SUBAPPLICATION Heckschieber (* Subapplication Type *)
  (* Standard: 61499-2 *)
  (* Version 1.0, 2023-01-29, Franz *)
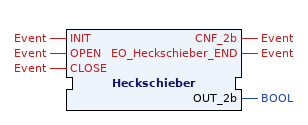
  EVENT_INPUT
    INIT;
    OPEN;
    CLOSE;
  END_EVENT
  EVENT_OUTPUT
    CNF_2b;
    EO_Heckschieber_END;
  END_EVENT
  VAR_OUTPUT
    OUT_2b : BOOL;
  END_VAR
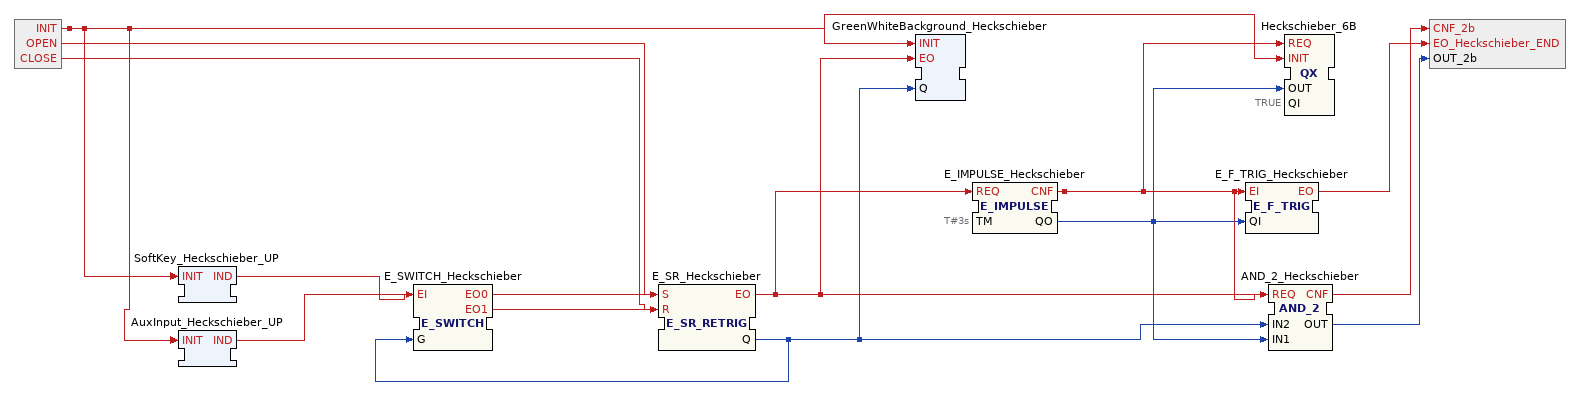
  FBS
    E_F_TRIG_Heckschieber : E_F_TRIG;
    Heckschieber_6B : QX(QI := TRUE);
    E_SR_Heckschieber : E_SR_RETRIG;
    E_SWITCH_Heckschieber : E_SWITCH;
    AND_2_Heckschieber : AND_2;
    E_IMPULSE_Heckschieber : E_IMPULSE(TM := T#3s);
  END_FBS
  SUBAPPLICATION AuxInput_Heckschieber_UP
    EVENT_INPUT
      INIT;
    END_EVENT
    EVENT_OUTPUT
      IND;
    END_EVENT
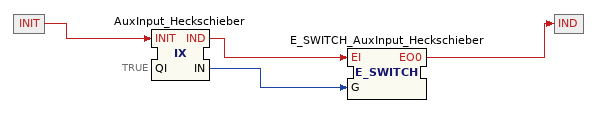
    FBS
      E_SWITCH_AuxInput_Heckschieber : E_SWITCH;
      AuxInput_Heckschieber : IX(QI := TRUE);
    END_FBS
    EVENT_CONNECTIONS
      AuxInput_Heckschieber.IND TO E_SWITCH_AuxInput_Heckschieber.EI;
      INIT TO AuxInput_Heckschieber.INIT;
      E_SWITCH_AuxInput_Heckschieber.EO0 TO IND;
    END_CONNECTIONS
    DATA_CONNECTIONS
      AuxInput_Heckschieber.IN TO E_SWITCH_AuxInput_Heckschieber.G;
    END_CONNECTIONS
  END_SUBAPPLICATION
  SUBAPPLICATION GreenWhiteBackground_Heckschieber
    EVENT_INPUT
      INIT;
      EO;
    END_EVENT
    VAR_INPUT
      Q : BOOL;
    END_VAR
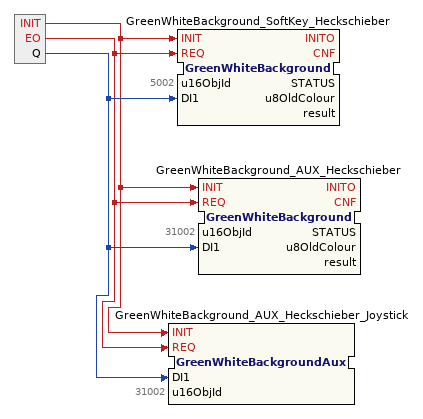
    FBS
      GreenWhiteBackground_SoftKey_Heckschieber : GreenWhiteBackground(u16ObjId := 5002);
      GreenWhiteBackground_AUX_Heckschieber : GreenWhiteBackground(u16ObjId := 31002);
      GreenWhiteBackground_AUX_Heckschieber_Joystick : GreenWhiteBackgroundAux(u16ObjId := 31002);
    END_FBS
    EVENT_CONNECTIONS
      INIT TO GreenWhiteBackground_SoftKey_Heckschieber.INIT;
      EO TO GreenWhiteBackground_SoftKey_Heckschieber.REQ;
      INIT TO GreenWhiteBackground_AUX_Heckschieber.INIT;
      EO TO GreenWhiteBackground_AUX_Heckschieber.REQ;
      INIT TO GreenWhiteBackground_AUX_Heckschieber_Joystick.INIT;
      EO TO GreenWhiteBackground_AUX_Heckschieber_Joystick.REQ;
    END_CONNECTIONS
    DATA_CONNECTIONS
      Q TO GreenWhiteBackground_SoftKey_Heckschieber.DI1;
      Q TO GreenWhiteBackground_AUX_Heckschieber.DI1;
      Q TO GreenWhiteBackground_AUX_Heckschieber_Joystick.DI1;
    END_CONNECTIONS
  END_SUBAPPLICATION
  SUBAPPLICATION SoftKey_Heckschieber_UP
    EVENT_INPUT
      INIT;
    END_EVENT
    EVENT_OUTPUT
      IND;
    END_EVENT
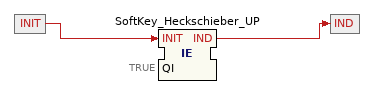
    FBS
      SoftKey_Heckschieber_UP : IE(QI := TRUE);
    END_FBS
    EVENT_CONNECTIONS
      INIT TO SoftKey_Heckschieber_UP.INIT;
      SoftKey_Heckschieber_UP.IND TO IND;
    END_CONNECTIONS
  END_SUBAPPLICATION
  EVENT_CONNECTIONS
    E_IMPULSE_Heckschieber.CNF TO E_F_TRIG_Heckschieber.EI;
    E_IMPULSE_Heckschieber.CNF TO Heckschieber_6B.REQ;
    E_SWITCH_Heckschieber.EO0 TO E_SR_Heckschieber.S;
    E_SWITCH_Heckschieber.EO1 TO E_SR_Heckschieber.R;
    E_SR_Heckschieber.EO TO AND_2_Heckschieber.REQ;
    E_SR_Heckschieber.EO TO E_IMPULSE_Heckschieber.REQ;
    E_IMPULSE_Heckschieber.CNF TO AND_2_Heckschieber.REQ;
    OPEN TO E_SR_Heckschieber.S;
    CLOSE TO E_SR_Heckschieber.R;
    AND_2_Heckschieber.CNF TO CNF_2b;
    E_F_TRIG_Heckschieber.EO TO EO_Heckschieber_END;
    AuxInput_Heckschieber_UP.IND TO E_SWITCH_Heckschieber.EI;
    INIT TO AuxInput_Heckschieber_UP.INIT;
    INIT TO GreenWhiteBackground_Heckschieber.INIT;
    E_SR_Heckschieber.EO TO GreenWhiteBackground_Heckschieber.EO;
    INIT TO SoftKey_Heckschieber_UP.INIT;
    SoftKey_Heckschieber_UP.IND TO E_SWITCH_Heckschieber.EI;
    INIT TO Heckschieber_6B.INIT;
  END_CONNECTIONS
  DATA_CONNECTIONS
    E_IMPULSE_Heckschieber.QO TO E_F_TRIG_Heckschieber.QI;
    E_IMPULSE_Heckschieber.QO TO Heckschieber_6B.OUT;
    E_SR_Heckschieber.Q TO E_SWITCH_Heckschieber.G;
    E_SR_Heckschieber.Q TO AND_2_Heckschieber.IN2;
    E_IMPULSE_Heckschieber.QO TO AND_2_Heckschieber.IN1;
    AND_2_Heckschieber.OUT TO OUT_2b;
    E_SR_Heckschieber.Q TO GreenWhiteBackground_Heckschieber.Q;
  END_CONNECTIONS
END_SUBAPPLICATION
